TYPE ST_CapManometer_CMR362 EXTENDS ST_VacuumGauge :
STRUCT
	rFull_Scale : REAL := 75.0 ;// Torr
END_STRUCT
END_TYPE

(* stored: Version 1.1.0.1, ProductVersion 3.1.4020.12
   DUT ST_CapManometer_CMR362: Id {e78f896f-852d-4bf0-a119-0ffe2d298eb2} *)
